DATA_BLOCK "DB2016_M_VF"
TITLE = DB2016_M_VF
{ S7_Optimized_Access := 'FALSE' }
AUTHOR : ABH
FAMILY : ZeusControl
VERSION : 1.0
//Bloque de datos motor variador.
   STRUCT
      M_VF { S7_SetPoint := 'False'} : Array[0.."N_MAX_DISP_M_VF"] of "UDT_ZC_DISP_M_VF";
      Mux { S7_SetPoint := 'False'} : Array[0.."N_MAX_MUX_DISP"] of "UDT_ZC_DISP_MUX_M_VF";
      Agrup : Array[0.."N_MAX_DISP_AGRUP"] of "UDT_ZC_DISP_AGRUP";
   END_STRUCT;


BEGIN
   M_VF[0].Hmi_Estado := 0;
   M_VF[0].Estado_Velocidad := 0.0;
   M_VF[0].Estado_AutoMan := FALSE;
   M_VF[0].Estado_Activado := FALSE;
   M_VF[0].Estado_Enclavado := FALSE;
   M_VF[0].Estado_EntradaTermico := FALSE;
   M_VF[0].Estado_EntradaConfMarcha := FALSE;
   M_VF[0].Alarmas_Termico := FALSE;
   M_VF[0].Alarmas_ConfirmacionMarcha := FALSE;
   M_VF[0].Alarmas_Mantenimiento := FALSE;
   M_VF[0].Alarmas_Escritura := FALSE;
   M_VF[0].Alarmas_Parametros := FALSE;
   M_VF[0].Alarmas_General := FALSE;
   M_VF[0].Orden_ActivarManual := FALSE;
   M_VF[0].Orden_ActivarAuto := FALSE;
   M_VF[0].Orden_ResetHoras := FALSE;
   M_VF[0].Config_Habilitar := FALSE;
   M_VF[0].Config_HabilitarRetornoTermico := TRUE;
   M_VF[0].Config_HabilitarInvertirTermico := FALSE;
   M_VF[0].Config_HabilitarRetornoConfMarcha := TRUE;
   M_VF[0].Config_HabilitarInvertirConfMarcha := FALSE;
   M_VF[0].Config_HabilitarMantenimiento := FALSE;
   M_VF[0].Config_HabilitarEscrituraSalida := FALSE;
   M_VF[0].Aux_oldActivado := FALSE;
   M_VF[0].Aux_oldAlarma := FALSE;
   M_VF[0].Aux_oldAutoMan := FALSE;
   M_VF[0].Estado_SeguridadOk := TRUE;
   M_VF[0].Config_GrupoAlarma := 0;
   M_VF[0].Estado_Escritura := 16#0000;
   M_VF[0].Orden_ConsignaManual := 0.0;
   M_VF[0].Orden_ConsignaAuto := 0.0;
   M_VF[0].Config_DireccionSalidaByte := 0;
   M_VF[0].Config_DireccionSalidaBit := 0;
   M_VF[0].Config_DireccionRetTermicoByte := 0;
   M_VF[0].Config_DireccionRetTermicoBit := 0;
   M_VF[0].Config_DireccionRetConfMarchaByte := 0;
   M_VF[0].Config_DireccionRetConfMarchaBit := 0;
   M_VF[0].Config_DireccionSalidaAnalogicaByte := 0;
   M_VF[0].Config_EscaladoMinIngenieria := 0.0;
   M_VF[0].Config_EscaladoMaxIngenieria := 50.0;
   M_VF[0].Tiempos_SetPointAlarma := 10;
   M_VF[0].Tiempos_Alarma := 0;
   M_VF[0].Tiempos_SetPointMantenimiento := 2000.0;
   M_VF[0].Tiempos_Mantenimiento := 0.0;
   M_VF[1].Hmi_Estado := 1;
   M_VF[1].Estado_Velocidad := 0.0;
   M_VF[1].Estado_AutoMan := FALSE;
   M_VF[1].Estado_Activado := FALSE;
   M_VF[1].Estado_Enclavado := FALSE;
   M_VF[1].Estado_EntradaTermico := FALSE;
   M_VF[1].Estado_EntradaConfMarcha := FALSE;
   M_VF[1].Alarmas_Termico := FALSE;
   M_VF[1].Alarmas_ConfirmacionMarcha := FALSE;
   M_VF[1].Alarmas_Mantenimiento := FALSE;
   M_VF[1].Alarmas_Escritura := FALSE;
   M_VF[1].Alarmas_Parametros := FALSE;
   M_VF[1].Alarmas_General := FALSE;
   M_VF[1].Orden_ActivarManual := FALSE;
   M_VF[1].Orden_ActivarAuto := FALSE;
   M_VF[1].Orden_ResetHoras := FALSE;
   M_VF[1].Config_Habilitar := TRUE;
   M_VF[1].Config_HabilitarRetornoTermico := TRUE;
   M_VF[1].Config_HabilitarInvertirTermico := TRUE;
   M_VF[1].Config_HabilitarRetornoConfMarcha := TRUE;
   M_VF[1].Config_HabilitarInvertirConfMarcha := FALSE;
   M_VF[1].Config_HabilitarMantenimiento := TRUE;
   M_VF[1].Config_HabilitarEscrituraSalida := TRUE;
   M_VF[1].Aux_oldActivado := FALSE;
   M_VF[1].Aux_oldAlarma := FALSE;
   M_VF[1].Aux_oldAutoMan := FALSE;
   M_VF[1].Estado_SeguridadOk := TRUE;
   M_VF[1].Config_GrupoAlarma := 0;
   M_VF[1].Estado_Escritura := 16#0000;
   M_VF[1].Orden_ConsignaManual := 95.0;
   M_VF[1].Orden_ConsignaAuto := 0.0;
   M_VF[1].Config_DireccionSalidaByte := 100;
   M_VF[1].Config_DireccionSalidaBit := 0;
   M_VF[1].Config_DireccionRetTermicoByte := 100;
   M_VF[1].Config_DireccionRetTermicoBit := 1;
   M_VF[1].Config_DireccionRetConfMarchaByte := 100;
   M_VF[1].Config_DireccionRetConfMarchaBit := 0;
   M_VF[1].Config_DireccionSalidaAnalogicaByte := 2100;
   M_VF[1].Config_EscaladoMinIngenieria := 0.0;
   M_VF[1].Config_EscaladoMaxIngenieria := 100.0;
   M_VF[1].Tiempos_SetPointAlarma := 10;
   M_VF[1].Tiempos_Alarma := 0;
   M_VF[1].Tiempos_SetPointMantenimiento := 2000.0;
   M_VF[1].Tiempos_Mantenimiento := 11.80547;
   Mux[0].Habilitar := TRUE;
   Mux[0].ExisteCambio := FALSE;
   Mux[0].MaxVisible := FALSE;
   Mux[0].Index := 5;
   Mux[0].oldIndex := 5;
   Mux[0].M_VF.Hmi_Estado := 1;
   Mux[0].M_VF.Estado_Velocidad := 0.0;
   Mux[0].M_VF.Estado_AutoMan := FALSE;
   Mux[0].M_VF.Estado_Activado := FALSE;
   Mux[0].M_VF.Estado_Enclavado := FALSE;
   Mux[0].M_VF.Estado_EntradaTermico := FALSE;
   Mux[0].M_VF.Estado_EntradaConfMarcha := FALSE;
   Mux[0].M_VF.Alarmas_Termico := FALSE;
   Mux[0].M_VF.Alarmas_ConfirmacionMarcha := FALSE;
   Mux[0].M_VF.Alarmas_Mantenimiento := FALSE;
   Mux[0].M_VF.Alarmas_Escritura := FALSE;
   Mux[0].M_VF.Alarmas_Parametros := FALSE;
   Mux[0].M_VF.Alarmas_General := FALSE;
   Mux[0].M_VF.Orden_ActivarManual := FALSE;
   Mux[0].M_VF.Orden_ActivarAuto := FALSE;
   Mux[0].M_VF.Orden_ResetHoras := FALSE;
   Mux[0].M_VF.Config_Habilitar := TRUE;
   Mux[0].M_VF.Config_HabilitarRetornoTermico := TRUE;
   Mux[0].M_VF.Config_HabilitarInvertirTermico := TRUE;
   Mux[0].M_VF.Config_HabilitarRetornoConfMarcha := TRUE;
   Mux[0].M_VF.Config_HabilitarInvertirConfMarcha := FALSE;
   Mux[0].M_VF.Config_HabilitarMantenimiento := FALSE;
   Mux[0].M_VF.Config_HabilitarEscrituraSalida := TRUE;
   Mux[0].M_VF.Aux_oldActivado := FALSE;
   Mux[0].M_VF.Aux_oldAlarma := FALSE;
   Mux[0].M_VF.Aux_oldAutoMan := FALSE;
   Mux[0].M_VF.Estado_SeguridadOk := TRUE;
   Mux[0].M_VF.Config_GrupoAlarma := 0;
   Mux[0].M_VF.Estado_Escritura := 16#0000;
   Mux[0].M_VF.Orden_ConsignaManual := 31.75312;
   Mux[0].M_VF.Orden_ConsignaAuto := 0.0;
   Mux[0].M_VF.Config_DireccionSalidaByte := 100;
   Mux[0].M_VF.Config_DireccionSalidaBit := 6;
   Mux[0].M_VF.Config_DireccionRetTermicoByte := 101;
   Mux[0].M_VF.Config_DireccionRetTermicoBit := 3;
   Mux[0].M_VF.Config_DireccionRetConfMarchaByte := 101;
   Mux[0].M_VF.Config_DireccionRetConfMarchaBit := 2;
   Mux[0].M_VF.Config_DireccionSalidaAnalogicaByte := 2110;
   Mux[0].M_VF.Config_EscaladoMinIngenieria := 0.0;
   Mux[0].M_VF.Config_EscaladoMaxIngenieria := 100.0;
   Mux[0].M_VF.Tiempos_SetPointAlarma := 10;
   Mux[0].M_VF.Tiempos_Alarma := 0;
   Mux[0].M_VF.Tiempos_SetPointMantenimiento := 2000.0;
   Mux[0].M_VF.Tiempos_Mantenimiento := 12.90666;
   Mux[1].Habilitar := TRUE;
   Mux[1].ExisteCambio := FALSE;
   Mux[1].MaxVisible := FALSE;
   Mux[1].Index := 0;
   Mux[1].oldIndex := 0;
   Mux[1].M_VF.Hmi_Estado := 0;
   Mux[1].M_VF.Estado_Velocidad := 0.0;
   Mux[1].M_VF.Estado_AutoMan := FALSE;
   Mux[1].M_VF.Estado_Activado := FALSE;
   Mux[1].M_VF.Estado_Enclavado := FALSE;
   Mux[1].M_VF.Estado_EntradaTermico := FALSE;
   Mux[1].M_VF.Estado_EntradaConfMarcha := FALSE;
   Mux[1].M_VF.Alarmas_Termico := FALSE;
   Mux[1].M_VF.Alarmas_ConfirmacionMarcha := FALSE;
   Mux[1].M_VF.Alarmas_Mantenimiento := FALSE;
   Mux[1].M_VF.Alarmas_Escritura := FALSE;
   Mux[1].M_VF.Alarmas_Parametros := FALSE;
   Mux[1].M_VF.Alarmas_General := FALSE;
   Mux[1].M_VF.Orden_ActivarManual := FALSE;
   Mux[1].M_VF.Orden_ActivarAuto := FALSE;
   Mux[1].M_VF.Orden_ResetHoras := FALSE;
   Mux[1].M_VF.Config_Habilitar := FALSE;
   Mux[1].M_VF.Config_HabilitarRetornoTermico := TRUE;
   Mux[1].M_VF.Config_HabilitarInvertirTermico := FALSE;
   Mux[1].M_VF.Config_HabilitarRetornoConfMarcha := TRUE;
   Mux[1].M_VF.Config_HabilitarInvertirConfMarcha := FALSE;
   Mux[1].M_VF.Config_HabilitarMantenimiento := FALSE;
   Mux[1].M_VF.Config_HabilitarEscrituraSalida := FALSE;
   Mux[1].M_VF.Aux_oldActivado := FALSE;
   Mux[1].M_VF.Aux_oldAlarma := FALSE;
   Mux[1].M_VF.Aux_oldAutoMan := FALSE;
   Mux[1].M_VF.Estado_SeguridadOk := TRUE;
   Mux[1].M_VF.Config_GrupoAlarma := 0;
   Mux[1].M_VF.Estado_Escritura := 16#0000;
   Mux[1].M_VF.Orden_ConsignaManual := 0.0;
   Mux[1].M_VF.Orden_ConsignaAuto := 0.0;
   Mux[1].M_VF.Config_DireccionSalidaByte := 0;
   Mux[1].M_VF.Config_DireccionSalidaBit := 0;
   Mux[1].M_VF.Config_DireccionRetTermicoByte := 0;
   Mux[1].M_VF.Config_DireccionRetTermicoBit := 0;
   Mux[1].M_VF.Config_DireccionRetConfMarchaByte := 0;
   Mux[1].M_VF.Config_DireccionRetConfMarchaBit := 0;
   Mux[1].M_VF.Config_DireccionSalidaAnalogicaByte := 0;
   Mux[1].M_VF.Config_EscaladoMinIngenieria := 0.0;
   Mux[1].M_VF.Config_EscaladoMaxIngenieria := 50.0;
   Mux[1].M_VF.Tiempos_SetPointAlarma := 10;
   Mux[1].M_VF.Tiempos_Alarma := 0;
   Mux[1].M_VF.Tiempos_SetPointMantenimiento := 2000.0;
   Mux[1].M_VF.Tiempos_Mantenimiento := 0.0;
   Agrup[0].AlgunaEnManual := FALSE;
   Agrup[0].AlgunaAlarma := FALSE;
   Agrup[0].NuevaAlarma := FALSE;
   Agrup[1].AlgunaEnManual := FALSE;
   Agrup[1].AlgunaAlarma := FALSE;
   Agrup[1].NuevaAlarma := FALSE;

END_DATA_BLOCK

